PROGRAM MAIN
VAR
END_VAR

P_Inputs();
P_Filtering();
P_ControlBlock();
P_Output();
//P_RunClock();
P_Modes();
P_PID();
P_FeedForward();

END_PROGRAM

(* stored: Version 1.1.0.1
   POU MAIN: Id {95bd3131-5c67-452d-927e-7536941f7837}, SpecialFunc None *)
